(* WARNING: This file is auto-generated. Do not modify it.*)
FUNCTION_BLOCK {{ fb_name }}
VAR_INPUT
    sTableName : STRING;
    {{ lookup_input }} : {{data_type}};
END_VAR
VAR_OUTPUT
{%- for output in outputs %}
    {{ output }} : {{ data_type }};
{%- endfor %}
    bError : BOOL; (* Was the table name or data invalid? *)
    bFound : BOOL; (* Was the input found in the table? *)
    bDone : BOOL;  (* Has the FB finished? *)

    fTableLookupLow: {{data_type}}; (* The lowest accepted lookup value. *)
    fTableLookupHigh: {{data_type}}; (* The highest accepted lookup value. *)
END_VAR
VAR

    bInit : BOOL;
    iRowSize : UDINT;
    fRow1 : POINTER TO ARRAY[0..{{ tables[0].bounds[1] }}] OF LREAL;
    fRow2 : POINTER TO ARRAY[0..{{ tables[0].bounds[1] }}] OF LREAL;
    {{ row_delta }} : {{data_type}};
    
    iRowCount : UDINT;
    iRowIdx : UDINT;
    fSlope : {{data_type}};

    (* The data tables. These are Initialized on the first function block call. *)
{% for table in tables %}
    {{table.name}} : ARRAY[{{table.indices_string}}] OF {{data_type}};
{% endfor %}
    
END_VAR


(* WARNING: This file is auto-generated. Do not modify it.*)

bError := FALSE;
bFound := FALSE;
bDone := FALSE;

IF NOT bInit THEN
{% for table in tables %}
    (* Table initialization: {{ table.name }} *)
    {{ table.data_as_code | indent(4) }}
{% endfor %}
    bInit := TRUE;
END_IF

(* Get correct table *)

{% for table in tables %}
{% if loop.index == 1 %}IF{% else %}ELSIF{% endif %} sTableName = '{{ table.identifier }}' THEN
    iRowSize := ADR({{ table.name }}[1,0]) - ADR({{ table.name }}[0,0]);
    iRowCount := {{ table.bounds[0] }};
    fRow1 := ADR({{ table.name }}[0, 0]);
    fTableLookupLow := {{ table.df.iloc[0, lookup_index] }};
    fTableLookupHigh := {{ table.df.iloc[-1, lookup_index] }};
{%- endfor %}
ELSE
    bError := TRUE;
    bDone := TRUE;
    RETURN;
END_IF

IF {{ lookup_input }} < fTableLookupLow THEN
    bDone := TRUE;
    RETURN;
ELSIF {{ lookup_input }} > fTableLookupHigh THEN
    bDone := TRUE;
    RETURN;
END_IF

FOR iRowIdx := 0 TO iRowCount - 1
DO
    fRow2 := fRow1 + iRowSize;
    IF {{ lookup_input }} >= fRow1^[{{ lookup_index }}] AND {{ lookup_input }} <= fRow2^[{{ lookup_index }}] THEN
        {{ row_delta }} := fRow2^[{{ lookup_index }}] - fRow1^[{{ lookup_index }}];
        IF {{ row_delta }} <= 0.0 THEN
            bFound := TRUE;
            bError := TRUE;
            bDone := TRUE;
        ELSE
{% for output in outputs %}
            // Interpolate output: {{ output }}
            fSlope := (fRow2^[{{ loop.index }}] - fRow1^[{{ loop.index }}]) / {{ row_delta }};
            {{ output }} := fRow1^[{{ loop.index}}] + fSlope * ({{ lookup_input }} - fRow1^[{{ lookup_index }}]);
{% endfor %} 
            bFound := TRUE;
            bError := FALSE;
            bDone := TRUE;
        END_IF
        RETURN;
    END_IF
    fRow1 := fRow2;
END_FOR

END_FUNCTION_BLOCK

(* stored: Version 1.1.0.1, ProductVersion 3.1.4024.4
   POU {{ fb_name }}: Id {{ '{' -}} {{ pou_guid }} {{- '}' }}, SpecialFunc None *)
